// Interface for a set implemented using a binary search tree.
INTERFACE I_Tree_Set EXTENDS I_Set

// Traversal method for retrieving values in the tree set.
PROPERTY _Traversal : T_BST_Traversal
GET
END_GET
SET
END_SET
END_PROPERTY

END_INTERFACE

(* stored: Version 1.1.0.1, ProductVersion 3.1.4024.4
   Itf I_Tree_Set: Id {739807ce-51a7-4ce0-ac23-8daf90e0493e}
   Property _Traversal: Id {d0dfd916-95e1-4892-9669-f9e9a8eb5bde}
   Get Get: Id {cff8a45c-267c-4474-b931-926165560000}
   Set Set: Id {59afb95d-dec8-4e13-b330-2cf4ec4792e8} *)
